// TIA Portal V20 export
TYPE "LER_typeRFIDCommands"
// stored: Access Published
   STRUCT
      readReq : Bool;
      writeReq : Bool;
      inventoryReq : Bool;
      ResetReq : Bool;
      resultRFIDReset : Bool;
   END_STRUCT;
END_TYPE
